// Edge cases of FB_EQ2HOR and FB_HOR2EQ: the celestial poles, an observer at a pole and on the equator, the zenith and
// the nadir, wrap-around of RA and azimuth, positions below the horizon and out-of-range angles.
//
// GENERATED by AstroBROT/testing/gen_block_tests.py from testing/golden_blocks.py, do not edit the numbers by hand.
// Every golden case is checked against the Python port of the ST (1E-7 deg) and against erfa (atco13 / atoc13) as a
// great-circle separation (2E-4 deg = 0.72 arcsec, no refraction, dut1 = 0). Altitude and azimuth are compared as a
// separation on the sky, not as two separate angle differences: near the zenith an azimuth difference is amplified by
// 1 / cos(alt) and says little about the pointing error (Azimuth_Difference_Is_Not_A_Sky_Separation).
FUNCTION_BLOCK FB_EdgeCases_Tests EXTENDS TcUnit.FB_TestSuite
VAR
END_VAR

EQ2HOR_North_celestial_pole();
EQ2HOR_South_celestial_pole();
EQ2HOR_RA_wrap_low();
EQ2HOR_RA_wrap_high();
EQ2HOR_Below_horizon();
EQ2HOR_Observer_at_north_pole();
EQ2HOR_Observer_at_south_pole();
EQ2HOR_Observer_on_equator();
HOR2EQ_Zenith_az0();
HOR2EQ_Zenith_az180();
HOR2EQ_Nadir();
HOR2EQ_Horizon_north();
HOR2EQ_Az_wrap_low();
HOR2EQ_Az_wrap_high();
HOR2EQ_Observer_at_north_pole();
HOR2EQ_Observer_at_south_pole();
HOR2EQ_Observer_on_equator();
HOR2EQ_Azimuth_Does_Not_Matter_At_The_Zenith();
HOR2EQ_Azimuth_Is_Periodic();
EQ2HOR_Right_Ascension_Is_Periodic();
EQ2HOR_Longitude_Is_Periodic();
EQ2HOR_Outputs_Stay_In_Range();
HOR2EQ_Outputs_Stay_In_Range();
Azimuth_Difference_Is_Not_A_Sky_Separation();

METHOD PRIVATE CheckNear
VAR_INPUT
	fExpected	: LREAL;
	fActual	: LREAL;
	fDelta	: LREAL;
	sName	: STRING(255);
END_VAR
AssertEquals_LREAL(Expected := fExpected, Actual := fActual, Delta := fDelta, Message := sName);
END_METHOD

METHOD PRIVATE CheckAngle
VAR_INPUT
	fExpected	: LREAL;
	fActual	: LREAL;
	fDelta	: LREAL;
	sName	: STRING(255);
END_VAR
VAR
	fDiff	: LREAL;
END_VAR
// angles in degrees, compared modulo 360 so that 359.9999999 and -1.0E-7 are equal
fDiff := fActual - fExpected;
WHILE fDiff > 180.0 DO fDiff := fDiff - 360.0; END_WHILE
WHILE fDiff < -180.0 DO fDiff := fDiff + 360.0; END_WHILE
AssertEquals_LREAL(Expected := 0.0, Actual := fDiff, Delta := fDelta, Message := sName);
END_METHOD

METHOD PRIVATE CheckSeparation
VAR_INPUT
	fLon1	: LREAL;
	fLat1	: LREAL;
	fLon2	: LREAL;
	fLat2	: LREAL;
	fDelta	: LREAL;
	sName	: STRING(255);
END_VAR
VAR
	fD2r	: LREAL;
	fHalfDLat	: LREAL;
	fHalfDLon	: LREAL;
	fHav	: LREAL;
	fSep	: LREAL;
END_VAR
// great-circle separation of two positions (longitude, latitude in degrees) against a tolerance in degrees;
// a difference of longitudes is not a distance on the sky, this is (haversine formula)
fD2r := 0.017453292519943295;
fHalfDLat := (fLat2 - fLat1) * fD2r * 0.5;
fHalfDLon := (fLon2 - fLon1) * fD2r * 0.5;
fHav := SIN(fHalfDLat) * SIN(fHalfDLat) + COS(fLat1 * fD2r) * COS(fLat2 * fD2r) * SIN(fHalfDLon) * SIN(fHalfDLon);
fSep := 2.0 * ASIN(SQRT(LIMIT(0.0, fHav, 1.0))) / fD2r;
AssertEquals_LREAL(Expected := 0.0, Actual := fSep, Delta := fDelta, Message := sName);
END_METHOD

METHOD PRIVATE EQ2HOR_North_celestial_pole
VAR
	fb	: AstroBROT.FB_EQ2HOR;
END_VAR
TEST('EQ2HOR_North_celestial_pole');
fb(ra := 0.0, dec := 90.0, jd := 2461300.75, lon := -16.5, lat := 28.3, refract := FALSE);
CheckNear(28.250439967419368, fb.alt, 1.0E-7, 'North_celestial_pole alt');
CheckAngle(0.15978772490399448, fb.az, 1.0E-7, 'North_celestial_pole az');
CheckSeparation(0.159877225222193, 28.250414281534653, fb.az, fb.alt, 0.0002, 'North_celestial_pole vs erfa');
TEST_FINISHED();
END_METHOD

METHOD PRIVATE EQ2HOR_South_celestial_pole
VAR
	fb	: AstroBROT.FB_EQ2HOR;
END_VAR
TEST('EQ2HOR_South_celestial_pole');
fb(ra := 0.0, dec := -90.0, jd := 2455197.5, lon := -70.7, lat := -30.2, refract := FALSE);
CheckNear(30.24486015624291, fb.alt, 1.0E-7, 'South_celestial_pole alt');
CheckAngle(180.02996665539834, fb.az, 1.0E-7, 'South_celestial_pole az');
CheckSeparation(180.02986430898196, 30.244862822992012, fb.az, fb.alt, 0.0002, 'South_celestial_pole vs erfa');
TEST_FINISHED();
END_METHOD

METHOD PRIVATE EQ2HOR_RA_wrap_low
VAR
	fb	: AstroBROT.FB_EQ2HOR;
END_VAR
TEST('EQ2HOR_RA_wrap_low');
fb(ra := 0.0001, dec := 22.01, jd := 2461300.75, lon := -16.5, lat := 28.3, refract := FALSE);
CheckNear(27.80734764100336, fb.alt, 1.0E-7, 'RA_wrap_low alt');
CheckAngle(281.5592750159755, fb.az, 1.0E-7, 'RA_wrap_low az');
CheckSeparation(281.55928456225905, 27.807403036183125, fb.az, fb.alt, 0.0002, 'RA_wrap_low vs erfa');
TEST_FINISHED();
END_METHOD

METHOD PRIVATE EQ2HOR_RA_wrap_high
VAR
	fb	: AstroBROT.FB_EQ2HOR;
END_VAR
TEST('EQ2HOR_RA_wrap_high');
fb(ra := 359.9999, dec := 22.01, jd := 2461300.75, lon := -16.5, lat := 28.3, refract := FALSE);
CheckNear(27.807174935931986, fb.alt, 1.0E-7, 'RA_wrap_high alt');
CheckAngle(281.55935130398774, fb.az, 1.0E-7, 'RA_wrap_high az');
CheckSeparation(281.5593608503559, 27.80723033089579, fb.az, fb.alt, 0.0002, 'RA_wrap_high vs erfa');
TEST_FINISHED();
END_METHOD

METHOD PRIVATE EQ2HOR_Below_horizon
VAR
	fb	: AstroBROT.FB_EQ2HOR;
END_VAR
TEST('EQ2HOR_Below_horizon');
fb(ra := 200.0, dec := -60.0, jd := 2461300.75, lon := -16.5, lat := 28.3, refract := FALSE);
CheckNear(-44.20054793244784, fb.alt, 1.0E-7, 'Below_horizon alt');
CheckAngle(148.24726062401623, fb.az, 1.0E-7, 'Below_horizon az');
CheckSeparation(148.2471745159021, -44.20052670358075, fb.az, fb.alt, 0.0002, 'Below_horizon vs erfa');
TEST_FINISHED();
END_METHOD

METHOD PRIVATE EQ2HOR_Observer_at_north_pole
VAR
	fb	: AstroBROT.FB_EQ2HOR;
END_VAR
TEST('EQ2HOR_Observer_at_north_pole');
fb(ra := 83.63, dec := 22.01, jd := 2461300.75, lon := 0.0, lat := 90.0, refract := FALSE);
CheckNear(22.028492329681235, fb.alt, 1.0E-7, 'Observer_at_north_pole alt');
CheckAngle(182.15756303104874, fb.az, 1.0E-7, 'Observer_at_north_pole az');
CheckSeparation(182.15754329791073, 22.028492563126676, fb.az, fb.alt, 0.0002, 'Observer_at_north_pole vs erfa');
TEST_FINISHED();
END_METHOD

METHOD PRIVATE EQ2HOR_Observer_at_south_pole
VAR
	fb	: AstroBROT.FB_EQ2HOR;
END_VAR
TEST('EQ2HOR_Observer_at_south_pole');
fb(ra := 83.63, dec := -22.01, jd := 2461300.75, lon := 0.0, lat := -90.0, refract := FALSE);
CheckNear(21.987455170067353, fb.alt, 1.0E-7, 'Observer_at_south_pole alt');
CheckAngle(357.7223600600331, fb.az, 1.0E-7, 'Observer_at_south_pole az');
CheckSeparation(357.7223798312026, 21.987453746489294, fb.az, fb.alt, 0.0002, 'Observer_at_south_pole vs erfa');
TEST_FINISHED();
END_METHOD

METHOD PRIVATE EQ2HOR_Observer_on_equator
VAR
	fb	: AstroBROT.FB_EQ2HOR;
END_VAR
TEST('EQ2HOR_Observer_on_equator');
fb(ra := 83.63, dec := 22.01, jd := 2461300.75, lon := -16.5, lat := 0.0, refract := FALSE);
CheckNear(63.91012183292501, fb.alt, 1.0E-7, 'Observer_on_equator alt');
CheckAngle(31.47678113024893, fb.az, 1.0E-7, 'Observer_on_equator az');
CheckSeparation(31.476987570998272, 63.910069653766755, fb.az, fb.alt, 0.0002, 'Observer_on_equator vs erfa');
TEST_FINISHED();
END_METHOD

METHOD PRIVATE HOR2EQ_Zenith_az0
VAR
	fb	: AstroBROT.FB_HOR2EQ;
END_VAR
TEST('HOR2EQ_Zenith_az0');
fb(alt := 90.0, az := 0.0, jd := 2461300.75, lon := -16.5, lat := 28.3, refract := FALSE);
CheckAngle(69.27121990661907, fb.ra, 1.0E-7, 'Zenith_az0 ra');
CheckNear(28.245793686130707, fb.dec, 1.0E-7, 'Zenith_az0 dec');
CheckSeparation(69.27111043655914, 28.245793175984534, fb.ra, fb.dec, 0.0002, 'Zenith_az0 vs erfa');
TEST_FINISHED();
END_METHOD

METHOD PRIVATE HOR2EQ_Zenith_az180
VAR
	fb	: AstroBROT.FB_HOR2EQ;
END_VAR
TEST('HOR2EQ_Zenith_az180');
fb(alt := 90.0, az := 180.0, jd := 2461300.75, lon := -16.5, lat := 28.3, refract := FALSE);
CheckAngle(69.27121990661907, fb.ra, 1.0E-7, 'Zenith_az180 ra');
CheckNear(28.245793686130707, fb.dec, 1.0E-7, 'Zenith_az180 dec');
CheckSeparation(69.27111043655914, 28.245793175984534, fb.ra, fb.dec, 0.0002, 'Zenith_az180 vs erfa');
TEST_FINISHED();
END_METHOD

METHOD PRIVATE HOR2EQ_Nadir
VAR
	fb	: AstroBROT.FB_HOR2EQ;
END_VAR
TEST('HOR2EQ_Nadir');
fb(alt := -90.0, az := 0.0, jd := 2461300.75, lon := -16.5, lat := 28.3, refract := FALSE);
CheckAngle(249.2743126674054, fb.ra, 1.0E-7, 'Nadir ra');
CheckNear(-28.244996713786396, fb.dec, 1.0E-7, 'Nadir dec');
CheckSeparation(249.27437964349747, -28.24499592575831, fb.ra, fb.dec, 0.0002, 'Nadir vs erfa');
TEST_FINISHED();
END_METHOD

METHOD PRIVATE HOR2EQ_Horizon_north
VAR
	fb	: AstroBROT.FB_HOR2EQ;
END_VAR
TEST('HOR2EQ_Horizon_north');
fb(alt := 0.0, az := 0.0, jd := 2461300.75, lon := -16.5, lat := 28.3, refract := FALSE);
CheckAngle(249.60995502319435, fb.ra, 1.0E-7, 'Horizon_north ra');
CheckNear(61.7487089558397, fb.dec, 1.0E-7, 'Horizon_north dec');
CheckSeparation(249.61009729239348, 61.74870711776769, fb.ra, fb.dec, 0.0002, 'Horizon_north vs erfa');
TEST_FINISHED();
END_METHOD

METHOD PRIVATE HOR2EQ_Az_wrap_low
VAR
	fb	: AstroBROT.FB_HOR2EQ;
END_VAR
TEST('HOR2EQ_Az_wrap_low');
fb(alt := 45.0, az := 0.0001, jd := 2461300.75, lon := -16.5, lat := 28.3, refract := FALSE);
CheckAngle(68.88002145549598, fb.ra, 1.0E-7, 'Az_wrap_low ra');
CheckNear(73.24907291497094, fb.dec, 1.0E-7, 'Az_wrap_low dec');
CheckSeparation(68.8797303761049, 73.24907332545713, fb.ra, fb.dec, 0.0002, 'Az_wrap_low vs erfa');
TEST_FINISHED();
END_METHOD

METHOD PRIVATE HOR2EQ_Az_wrap_high
VAR
	fb	: AstroBROT.FB_HOR2EQ;
END_VAR
TEST('HOR2EQ_Az_wrap_high');
fb(alt := 45.0, az := 359.9999, jd := 2461300.75, lon := -16.5, lat := 28.3, refract := FALSE);
CheckAngle(68.87953075699878, fb.ra, 1.0E-7, 'Az_wrap_high ra');
CheckNear(73.24907170989893, fb.dec, 1.0E-7, 'Az_wrap_high dec');
CheckSeparation(68.87923967758073, 73.2490721197454, fb.ra, fb.dec, 0.0002, 'Az_wrap_high vs erfa');
TEST_FINISHED();
END_METHOD

METHOD PRIVATE HOR2EQ_Observer_at_north_pole
VAR
	fb	: AstroBROT.FB_HOR2EQ;
END_VAR
TEST('HOR2EQ_Observer_at_north_pole');
fb(alt := 40.0, az := 100.0, jd := 2461300.75, lon := 0.0, lat := 90.0, refract := FALSE);
CheckAngle(165.82212182028053, fb.ra, 1.0E-7, 'Observer_at_north_pole ra');
CheckNear(40.14345354944047, fb.dec, 1.0E-7, 'Observer_at_north_pole dec');
CheckSeparation(165.82210357343894, 40.14345009010985, fb.ra, fb.dec, 0.0002, 'Observer_at_north_pole vs erfa');
TEST_FINISHED();
END_METHOD

METHOD PRIVATE HOR2EQ_Observer_at_south_pole
VAR
	fb	: AstroBROT.FB_HOR2EQ;
END_VAR
TEST('HOR2EQ_Observer_at_south_pole');
fb(alt := -20.0, az := 100.0, jd := 2461300.75, lon := 0.0, lat := -90.0, refract := FALSE);
CheckAngle(185.85805478189764, fb.ra, 1.0E-7, 'Observer_at_south_pole ra');
CheckNear(20.14661753333691, fb.dec, 1.0E-7, 'Observer_at_south_pole dec');
CheckSeparation(185.85803179512064, 20.146612025652036, fb.ra, fb.dec, 0.0002, 'Observer_at_south_pole vs erfa');
TEST_FINISHED();
END_METHOD

METHOD PRIVATE HOR2EQ_Observer_on_equator
VAR
	fb	: AstroBROT.FB_HOR2EQ;
END_VAR
TEST('HOR2EQ_Observer_on_equator');
fb(alt := 60.0, az := 250.0, jd := 2461300.75, lon := -16.5, lat := 0.0, refract := FALSE);
CheckAngle(40.87970090453398, fb.ra, 1.0E-7, 'Observer_on_equator ra');
CheckNear(-9.963791072363595, fb.dec, 1.0E-7, 'Observer_on_equator dec');
CheckSeparation(40.879599464361846, -9.963785329026702, fb.ra, fb.dec, 0.0002, 'Observer_on_equator vs erfa');
TEST_FINISHED();
END_METHOD

METHOD PRIVATE HOR2EQ_Azimuth_Does_Not_Matter_At_The_Zenith
VAR
	fbA	: AstroBROT.FB_HOR2EQ;
	fbB	: AstroBROT.FB_HOR2EQ;
END_VAR
TEST('HOR2EQ_Azimuth_Does_Not_Matter_At_The_Zenith');
fbA(alt := 90.0, az := 0.0, jd := 2461300.75, lon := -16.5, lat := 28.3, refract := FALSE);
fbB(alt := 90.0, az := 180.0, jd := 2461300.75, lon := -16.5, lat := 28.3, refract := FALSE);
CheckAngle(fbA.ra, fbB.ra, 1.0E-9, 'ra');
CheckNear(fbA.dec, fbB.dec, 1.0E-9, 'dec');
AssertTrue(Condition := fbA.dec > 0.0 AND fbA.dec < 90.0, Message := 'the zenith of a northern site has 0 < dec < 90 (no NaN from ASIN)');
TEST_FINISHED();
END_METHOD

METHOD PRIVATE HOR2EQ_Azimuth_Is_Periodic
VAR
	fbRef	: AstroBROT.FB_HOR2EQ;
	fb	: AstroBROT.FB_HOR2EQ;
END_VAR
TEST('HOR2EQ_Azimuth_Is_Periodic');
fbRef(alt := 45.0, az := 350.0, jd := 2461300.75, lon := -16.5, lat := 28.3, refract := FALSE);
fb(alt := 45.0, az := -10.0, jd := 2461300.75, lon := -16.5, lat := 28.3, refract := FALSE);
CheckAngle(fbRef.ra, fb.ra, 1.0E-9, 'az -10 ra');
CheckNear(fbRef.dec, fb.dec, 1.0E-9, 'az -10 dec');
fb(alt := 45.0, az := 710.0, jd := 2461300.75, lon := -16.5, lat := 28.3, refract := FALSE);
CheckAngle(fbRef.ra, fb.ra, 1.0E-9, 'az 710 ra');
CheckNear(fbRef.dec, fb.dec, 1.0E-9, 'az 710 dec');
TEST_FINISHED();
END_METHOD

METHOD PRIVATE EQ2HOR_Right_Ascension_Is_Periodic
VAR
	fbRef	: AstroBROT.FB_EQ2HOR;
	fb	: AstroBROT.FB_EQ2HOR;
END_VAR
TEST('EQ2HOR_Right_Ascension_Is_Periodic');
fbRef(ra := 83.63, dec := 22.01, jd := 2461300.75, lon := -16.5, lat := 28.3, refract := FALSE);
fb(ra := -276.37, dec := 22.01, jd := 2461300.75, lon := -16.5, lat := 28.3, refract := FALSE);
CheckNear(fbRef.alt, fb.alt, 1.0E-9, 'ra -276.37 alt');
CheckAngle(fbRef.az, fb.az, 1.0E-9, 'ra -276.37 az');
fb(ra := 443.63, dec := 22.01, jd := 2461300.75, lon := -16.5, lat := 28.3, refract := FALSE);
CheckNear(fbRef.alt, fb.alt, 1.0E-9, 'ra 443.63 alt');
CheckAngle(fbRef.az, fb.az, 1.0E-9, 'ra 443.63 az');
TEST_FINISHED();
END_METHOD

METHOD PRIVATE EQ2HOR_Longitude_Is_Periodic
VAR
	fbRef	: AstroBROT.FB_EQ2HOR;
	fb	: AstroBROT.FB_EQ2HOR;
END_VAR
TEST('EQ2HOR_Longitude_Is_Periodic');
fbRef(ra := 83.63, dec := 22.01, jd := 2461300.75, lon := -16.5, lat := 28.3, refract := FALSE);
fb(ra := 83.63, dec := 22.01, jd := 2461300.75, lon := 343.5, lat := 28.3, refract := FALSE);
CheckNear(fbRef.alt, fb.alt, 1.0E-9, 'lon 343.5 alt');
CheckAngle(fbRef.az, fb.az, 1.0E-9, 'lon 343.5 az');
TEST_FINISHED();
END_METHOD

METHOD PRIVATE EQ2HOR_Outputs_Stay_In_Range
VAR
	fb	: AstroBROT.FB_EQ2HOR;
	i	: INT;
	fDec	: LREAL;
END_VAR
TEST('EQ2HOR_Outputs_Stay_In_Range');
// declinations from pole to pole for observers at both poles, on the equator and at a mid latitude
FOR i := -2 TO 2 DO
	fDec := 45.0 * i;
	fb(ra := 200.0, dec := fDec, jd := 2461300.75, lon := 0.0, lat := 90.0, refract := FALSE);
	AssertTrue(Condition := fb.alt >= -90.0 AND fb.alt <= 90.0 AND fb.az >= 0.0 AND fb.az <= 360.0, Message := 'observer at the north pole');
	fb(ra := 200.0, dec := fDec, jd := 2461300.75, lon := 0.0, lat := -90.0, refract := FALSE);
	AssertTrue(Condition := fb.alt >= -90.0 AND fb.alt <= 90.0 AND fb.az >= 0.0 AND fb.az <= 360.0, Message := 'observer at the south pole');
	fb(ra := 200.0, dec := fDec, jd := 2461300.75, lon := 0.0, lat := 0.0, refract := FALSE);
	AssertTrue(Condition := fb.alt >= -90.0 AND fb.alt <= 90.0 AND fb.az >= 0.0 AND fb.az <= 360.0, Message := 'observer on the equator');
	fb(ra := 200.0, dec := fDec, jd := 2461300.75, lon := -16.5, lat := 28.3, refract := FALSE);
	AssertTrue(Condition := fb.alt >= -90.0 AND fb.alt <= 90.0 AND fb.az >= 0.0 AND fb.az <= 360.0, Message := 'observer at 28.3 deg');
END_FOR
TEST_FINISHED();
END_METHOD

METHOD PRIVATE HOR2EQ_Outputs_Stay_In_Range
VAR
	fb	: AstroBROT.FB_HOR2EQ;
	i	: INT;
	fAlt	: LREAL;
END_VAR
TEST('HOR2EQ_Outputs_Stay_In_Range');
// altitudes from nadir to zenith, for observers at both poles, on the equator and at a mid latitude
FOR i := -2 TO 2 DO
	fAlt := 45.0 * i;
	fb(alt := fAlt, az := 100.0, jd := 2461300.75, lon := 0.0, lat := 90.0, refract := FALSE);
	AssertTrue(Condition := fb.dec >= -90.0 AND fb.dec <= 90.0 AND fb.ra >= 0.0 AND fb.ra < 360.0, Message := 'observer at the north pole');
	fb(alt := fAlt, az := 100.0, jd := 2461300.75, lon := 0.0, lat := -90.0, refract := FALSE);
	AssertTrue(Condition := fb.dec >= -90.0 AND fb.dec <= 90.0 AND fb.ra >= 0.0 AND fb.ra < 360.0, Message := 'observer at the south pole');
	fb(alt := fAlt, az := 100.0, jd := 2461300.75, lon := 0.0, lat := 0.0, refract := FALSE);
	AssertTrue(Condition := fb.dec >= -90.0 AND fb.dec <= 90.0 AND fb.ra >= 0.0 AND fb.ra < 360.0, Message := 'observer on the equator');
	fb(alt := fAlt, az := 100.0, jd := 2461300.75, lon := -16.5, lat := 28.3, refract := FALSE);
	AssertTrue(Condition := fb.dec >= -90.0 AND fb.dec <= 90.0 AND fb.ra >= 0.0 AND fb.ra < 360.0, Message := 'observer at 28.3 deg');
END_FOR
TEST_FINISHED();
END_METHOD

METHOD PRIVATE Azimuth_Difference_Is_Not_A_Sky_Separation
VAR
	fb1	: AstroBROT.FB_EQ2HOR;
	fb2	: AstroBROT.FB_EQ2HOR;
	fAzDiff	: LREAL;
END_VAR
TEST('Azimuth_Difference_Is_Not_A_Sky_Separation');
// The review recorded "azimuth outliers up to 40 arcsec" as a coordinate difference. Two positions 0.63 arcsec apart on the sky
// (0.05 deg from the zenith) differ by 629 arcsec in azimuth: the azimuth difference is amplified by 1 / cos(alt) = 1146.
// A raw azimuth difference therefore cannot be used as an accuracy figure; a great-circle separation can.
fb1(ra := 69.29947685614172, dec := 28.289165400359746, jd := 2461300.75, lon := -16.5, lat := 28.3, refract := FALSE);
fb2(ra := 69.29967685614173, dec := 28.289165400359746, jd := 2461300.75, lon := -16.5, lat := 28.3, refract := FALSE);
fAzDiff := fb2.az - fb1.az;
CheckNear(0.17470443800883118, fAzDiff, 1.0E-6, 'azimuth difference in degrees');
CheckSeparation(fb1.az, fb1.alt, fb2.az, fb2.alt, 0.00017709654618499777, 'separation of the two outputs is the sky separation');
AssertTrue(Condition := ABS(fAzDiff) > 100.0 * 0.00017609654618499777, Message := 'the azimuth difference is more than 100 times the separation');
TEST_FINISHED();
END_METHOD

END_FUNCTION_BLOCK

(* stored: Version 1.1.0.1, ProductVersion 3.1.4024.15
   POU FB_EdgeCases_Tests: Id {1ce8b4dd-f252-5622-aeba-d16d757419d4}, SpecialFunc None
   Method CheckNear: Id {ae5cbb73-9f17-5456-abe9-3e9b636050b5}
   Method CheckAngle: Id {fd336346-3738-5635-b78e-b47f4140cf69}
   Method CheckSeparation: Id {831c8b0c-dd19-532e-b7cc-0fd2562e4b20}
   Method EQ2HOR_North_celestial_pole: Id {95d3a9f0-640d-5335-ba09-ca793b23a8b8}
   Method EQ2HOR_South_celestial_pole: Id {0a166255-24b3-5f7a-b863-4a67b1e05c86}
   Method EQ2HOR_RA_wrap_low: Id {02389d38-67d9-5fdf-9eae-3aa7d42942ba}
   Method EQ2HOR_RA_wrap_high: Id {080d1fc2-74a5-5dc2-bd95-55185a94e1b2}
   Method EQ2HOR_Below_horizon: Id {de2d3df4-2d17-5a5f-b60d-ff726ff706cb}
   Method EQ2HOR_Observer_at_north_pole: Id {321f7bfb-8ed9-56c3-9b39-4ee6022a1482}
   Method EQ2HOR_Observer_at_south_pole: Id {9309b22c-e8bc-5b3f-86c5-34bbfb5f254f}
   Method EQ2HOR_Observer_on_equator: Id {9cd88f17-fea6-5dd8-8073-a6c8e9c8e5e6}
   Method HOR2EQ_Zenith_az0: Id {05ca6b99-2977-5e01-853a-c046afc1d25a}
   Method HOR2EQ_Zenith_az180: Id {bb54b10b-8dfe-564f-aba5-52f007283402}
   Method HOR2EQ_Nadir: Id {ae0eae25-8b99-536d-9518-ac4dd821af68}
   Method HOR2EQ_Horizon_north: Id {74e1bf8a-b5a2-5399-81d5-c8ec49610ecb}
   Method HOR2EQ_Az_wrap_low: Id {c1ed5c4a-9271-540d-8dc2-cba7c010facd}
   Method HOR2EQ_Az_wrap_high: Id {9cbd6a23-dd83-5c0c-a811-7b4074b40716}
   Method HOR2EQ_Observer_at_north_pole: Id {dc7838b1-6e79-5f5a-8fdd-94cb81b3fe2e}
   Method HOR2EQ_Observer_at_south_pole: Id {b464d2a6-bd48-5ca2-94a3-a7f73d60a054}
   Method HOR2EQ_Observer_on_equator: Id {f77bc31c-dc21-534b-beb8-dde3c93cd236}
   Method HOR2EQ_Azimuth_Does_Not_Matter_At_The_Zenith: Id {44d9fe50-648f-51d0-8226-c10a05a2a39f}
   Method HOR2EQ_Azimuth_Is_Periodic: Id {99b74d67-2a2c-5b07-986a-244312c2c69c}
   Method EQ2HOR_Right_Ascension_Is_Periodic: Id {802adb4c-87c0-54df-b7b7-12df75e586ed}
   Method EQ2HOR_Longitude_Is_Periodic: Id {ec0685f9-9ae2-5512-8a76-bad041ff1830}
   Method EQ2HOR_Outputs_Stay_In_Range: Id {30c9487b-2186-5374-94c0-383dbeb4b040}
   Method HOR2EQ_Outputs_Stay_In_Range: Id {ad1345e8-9e47-5666-bbb8-5f56a69c4da0}
   Method Azimuth_Difference_Is_Not_A_Sky_Separation: Id {1e01fdc4-d0df-561a-b0d1-30486cfa78ce} *)
